(* PLC project SansNom, Inconnu SansNom 1 *)
(* stored: creationDateTime 2025-01-02T16:30:26, modificationDateTime 2025-01-09T15:00:52 *)

PROGRAM hello_world
  VAR
    A : BOOL := true;
    B : BOOL := false;
    C : BOOL;
    O : BOOL;
  END_VAR

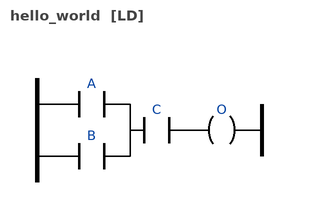
(* LD diagram, written out as Structured Text *)
O := (B OR A) AND C;
END_PROGRAM

CONFIGURATION Config0
  RESOURCE Res0 ON PLC
    TASK task0(INTERVAL := T#20ms, PRIORITY := 0);
    PROGRAM instance0 WITH task0 : hello_world;
  END_RESOURCE
END_CONFIGURATION
